// TIA Portal V17 export
// export: Created 2026-07-06T15:33:03.2786361Z, ExportSetting WithDefaults, DisplayName Totally Integrated Automation Portal, DisplayVersion V17, DisplayName TIA Portal Openness, DisplayVersion V17, DisplayName TIA Portal Version Control Interface, DisplayVersion V17, DisplayName STEP 7 Professional, DisplayVersion V17, DisplayName STEP 7 Safety, DisplayVersion V17, DisplayName WinCC Professional, DisplayVersion V17
FUNCTION_BLOCK "Canet_com"   // FB3, LAD
{ S7_Optimized_Access := 'FALSE' }
VERSION : 0.1
// stored: AutoNumber true, IsIECCheckEnabled false, SetENOAutomatically false, UDAEnableTagReadback false
   VAR_INPUT
      con_req : Bool;
   END_VAR
   VAR_OUTPUT
      connection_established : Bool;
   END_VAR
   VAR_IN_OUT
      Data_rcvd : Array[0..12] of Byte;
   END_VAR
BEGIN

REGION Network 1: Connection
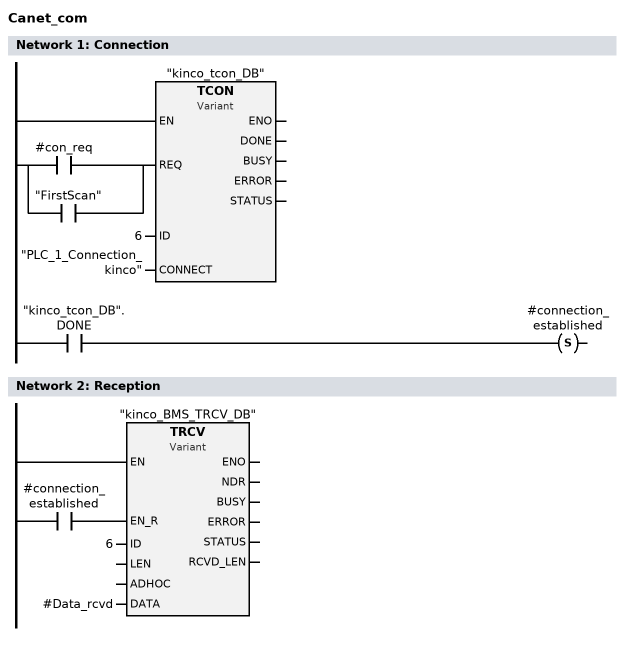
   RUNG wire#powerrail
      { S7_Templates := "[con_type := Variant, id_type := CONN_OUC]" } "kinco_tcon_DB".TCON(REQ := wire#w1, ID := 6, CONNECT := "PLC_1_Connection_kinco", DONE =>, BUSY =>, ERROR =>, STATUS =>)
   END_RUNG
   RUNG wire#powerrail
      Contact( #con_req )
   END_RUNG wire#w1
   RUNG wire#powerrail
      Contact( "FirstScan" )
   END_RUNG wire#w1
   RUNG wire#powerrail
      Contact( "kinco_tcon_DB".DONE )
      S_Coil( #connection_established )
   END_RUNG
   // the same network as SCL:
   "kinco_tcon_DB"(REQ := #con_req OR "FirstScan", ID := 6, CONNECT := "PLC_1_Connection_kinco");   // TCON
   IF "kinco_tcon_DB".DONE THEN #connection_established := TRUE; END_IF;
END_REGION

REGION Network 2: Reception
   RUNG wire#powerrail
      { S7_Templates := "[card := 1, ptr_type := Variant, value_type := UDInt, id_type := CONN_OUC]" } "kinco_BMS_TRCV_DB".TRCV(EN_R := wire#w1, ID := 6, LEN :=, ADHOC :=, DATA := #Data_rcvd, NDR =>, BUSY =>, ERROR =>, STATUS =>, RCVD_LEN =>)
   END_RUNG
   RUNG wire#powerrail
      Contact( #connection_established )
   END_RUNG wire#w1
   // the same network as SCL:
   "kinco_BMS_TRCV_DB"(EN_R := #connection_established, ID := 6, DATA := #Data_rcvd);   // TRCV
END_REGION
END_FUNCTION_BLOCK
